TYPE ST_DCLink_IO :
STRUCT
	bMCCBOpen		AT %Q*: BOOL;
	bMCCBClose		AT %Q*: BOOL;
	bUVRfb			AT %I*: BOOL;
END_STRUCT
END_TYPE

(* stored: Version 1.1.0.1, ProductVersion 3.1.4026.18
   DUT ST_DCLink_IO: Id {024d705a-f584-43ee-b9ef-f67055b7fe29} *)
